(* IEC 61131-3 sources: POMIRTS_lab3/AS/Library/FB_lib, 3 files *)

(* ---- FB_lib.typ ---- *)
(********************************************************************
 * COPYRIGHT -- Bernecker + Rainer
 ********************************************************************
 * Library: FB_lib
 * File: FB_lib.typ
 * Author: B+R
 ********************************************************************
 * Data types of library FB_lib
 ********************************************************************)

TYPE
	FBDevice_typ : STRUCT			(*internal use*)
		MemorySize	: USINT ;
		DevAdress	: UDINT ;
		DevInfo	: UDINT ;
		Error	: UINT ;
		FBIdent	: UDINT ;
		DevNumber	: UINT ;
		DevType	: USINT ;
		ConfMsgNr	: USINT ;
		CommandMsgNr	: USINT ;
		StatusMsgNr	: USINT ;
		OtherMsgNr	: USINT ;
	END_STRUCT;
END_TYPE

(* ---- FB_lib.fun ---- *)
(********************************************************************
 * COPYRIGHT -- Bernecker + Rainer
 ********************************************************************
 * Library: FB_lib
 * File: FB_lib.fun
 * Author: B+R
 ********************************************************************
 * Functions and function blocks of library FB_lib
 ********************************************************************)

FUNCTION_BLOCK FBio					(*copies the input and output data areas between the B&R card and the specified buffers; asynchronous execution*)
	VAR_INPUT
		enable	:BOOL;				(*enables execution*)
		DevIdent	:UDINT;			(*device identifier returned from FBInit*)
		OutBuffer	:UDINT;			(*pointer to the output data area*)
		OutLen	:UDINT;				(*length of the output data area*)
		InBuffer	:UDINT;			(*pointer to the input data area*)
		InLen	:UDINT;				(*length of the input data area*)
	END_VAR
	VAR_OUTPUT
		status	:UINT;				(*execution status: ERR_OK, ERR_FUB_ENABLE_FALSE, ERR_FUB_BUSY, 0xXXXX = see help*)
	END_VAR
	VAR
		hmode	:USINT;				(*internal variable*)
	END_VAR
END_FUNCTION_BLOCK

FUNCTION_BLOCK FBStart				(*starts the I/O exchange process*)
	VAR_INPUT
		enable	:BOOL;				(*enables execution*)
		DevIdent	:UDINT;			(*device identifier returned from FBInit*)
	END_VAR
	VAR_OUTPUT
		status	:UINT;				(*execution status: ERR_OK, ERR_FUB_ENABLE_FALSE, 0xXXXX = see help*)
	END_VAR
END_FUNCTION_BLOCK

FUNCTION_BLOCK FBStop				(*stops the I/O exchange process*)
	VAR_INPUT
		enable	:BOOL;				(*enables execution*)
		DevIdent	:UDINT;			(*device identifier returned from FBInit*)
	END_VAR
	VAR_OUTPUT
		status	:UINT;				(*execution status: ERR_OK, ERR_FUB_ENABLE_FALSE, 0xXXXX = see help*)
	END_VAR
END_FUNCTION_BLOCK

FUNCTION_BLOCK FBSlaveStat			(*returns the current slave status*)
	VAR_INPUT
		enable	:BOOL;				(*enables execution*)
		DevIdent	:UDINT;			(*device identifier returned from FBInit*)
		SlaveReady	:UDINT;			(*pointer to a 16 byte array indicating whether a slave is in data transfer mode*)
		SlaveDiag	:UDINT;			(*pointer to a 16 byte array indicating the availability of diagnose information on slaves*)
	END_VAR
	VAR_OUTPUT
		status	:UINT;				(*execution status: ERR_OK, ERR_FUB_ENABLE_FALSE, 0xXXXX = see help*)
		SlaveStatus	:BOOL;			(*TRUE = a configured slave is not in data transfer mode or has diagnostic messages*)
	END_VAR
END_FUNCTION_BLOCK

FUNCTION_BLOCK FBInit				(*searches and initializes the specified device*)
	VAR_INPUT
		enable	:BOOL;				(*enables execution*)
		Device	:UDINT;				(*device name given as pointer, e.g., "SL2.SS1.IF1"*)
	END_VAR
	VAR_OUTPUT
		status	:UINT;				(*execution status: ERR_OK, ERR_FUB_ENABLE_FALSE, 0xXXXX = see help*)
		MemSize	:USINT;				(*indicates the FB size on the card*)
		DevIdent	:UDINT;			(*device identifier*)
		Run	:BOOL;					(*device in run: TRUE = in run, FALSE = not in run*)
		Configuration	:BOOL;		(*configuration: TRUE = valid, FALSE = not valid*)
	END_VAR
END_FUNCTION_BLOCK

FUNCTION_BLOCK FBSlaveExtStat		(*returns the exact status of a slave; asynchronous execution*)
	VAR_INPUT
		enable	:BOOL;				(*enables execution*)
		DevIdent	:UDINT;			(*device identifier returned from FBInit*)
		SlaveNumber	:USINT;			(*slave number*)
		SlaveDiagnostic	:UDINT;		(*pointer to an array of 48 bytes containing extended status and diagnostic information*)
	END_VAR
	VAR_OUTPUT
		status	:UINT;				(*execution status: ERR_OK, ERR_FUB_ENABLE_FALSE, ERR_FUB_BUSY, 0xXXXX = see help*)
		SlaveReady	:BOOL;			(*TRUE = slave is not in data transfer mode*)
		SlaveDiag	:BOOL;			(*TRUE = slave is in diagnostics mode*)
	END_VAR
	VAR
		istate	:UDINT;				(*internal variable*)
		waitCnt	:UINT;				(*internal variable*)
	END_VAR
END_FUNCTION_BLOCK

FUNCTION_BLOCK FBConfig				(*downloads the configuration; asynchronous execution*)
	VAR_INPUT
		enable	:BOOL;				(*enables execution*)
		DevIdent	:UDINT;			(*device identifier returned from FBInit*)
		ConfModulName	:UDINT;		(*configuration module name given as pointer*)
		Mode	:BOOL;				(*download mode, TRUE = sequential, FALSE = in one step*)
	END_VAR
	VAR_OUTPUT
		status	:UINT;				(*execution status: ERR_OK, ERR_FUB_ENABLE_FALSE, ERR_FUB_BUSY, 0xXXXX = see help*)
		Remaining	:UDINT;			(*displays the remaining segments until the configuration is completely loaded*)
	END_VAR
	VAR
		istate	:UDINT;				(*internal variable*)
		FileLength	:UINT;			(*internal variable*)
		waitCnt	:UINT;				(*internal variable*)
		OffsetCopy	:UDINT;			(*internal variable*)
		pData	:UDINT;				(*internal variable*)
		Ready	:USINT;				(*internal variable*)
		FirstMessage	:BOOL;		(*internal variable*)
		MsgPutReady	:BOOL;			(*internal variable*)
	END_VAR
END_FUNCTION_BLOCK

FUNCTION_BLOCK FBDialog				(*send messages to the B&R card; asynchronous execution*)
	VAR_INPUT
		enable	:BOOL;				(*enables execution*)
		DevIdent	:UDINT;			(*device identifier returned from FBInit*)
		Message	:UDINT;				(*pointer to the message structure*)
	END_VAR
	VAR_OUTPUT
		status	:UINT;				(*execution status: ERR_OK, ERR_FUB_ENABLE_FALSE, ERR_FUB_BUSY, 0xXXXX = see help*)
	END_VAR
	VAR
		istate	:UDINT;				(*internal variable*)
		tx	:USINT;					(*internal variable*)
		waitCount	:UINT;			(*internal variable*)
	END_VAR
END_FUNCTION_BLOCK

FUNCTION FBSearchDevices : UINT		(*searches the target system for B&R fieldbus cards*)
	VAR_INPUT
		pInfos	:UDINT;				(*pointer to the device information structure*)
		count	:USINT;				(*number of devices to be searched*)
	END_VAR
END_FUNCTION

FUNCTION_BLOCK FBGetMessage           (*sends a message to the B&R card and does not wait for an answer; asynchronous execution*)
	VAR_INPUT
		enable	:BOOL;                 (*enables execution*)
		DevIdent	:UDINT;            (*device identifier returned from DPMInit*)
		Message	:UDINT;                (*pointer to the message structure*)
	END_VAR
	VAR_OUTPUT
		status	:UINT;                 (*execution status: ERR_OK, ERR_FUB_ENABLE_FALSE, ERR_FUB_BUSY, 0xXXXX = see help*)
	END_VAR
	VAR
		waitCount	:UINT;             (*internal variable*)
	END_VAR
END_FUNCTION_BLOCK

FUNCTION_BLOCK FBPutMessage            (*reads out a message from the B&R card; asynchronous execution*)
	VAR_INPUT
		enable	:BOOL;                 (*enables execution*)
		DevIdent	:UDINT;            (*device identifier returned from DPMInit*)
		Message	:UDINT;                (*pointer to the message structure*)
	END_VAR
	VAR_OUTPUT
		status	:UINT;                 (*execution status: ERR_OK, ERR_FUB_ENABLE_FALSE, ERR_FUB_BUSY, 0xXXXX = see help*)
	END_VAR
	VAR
		waitCount	:UINT;             (*internal variable*)
	END_VAR
END_FUNCTION_BLOCK

(* ---- FB_lib.var ---- *)
(********************************************************************
 * COPYRIGHT -- Bernecker + Rainer
 ********************************************************************
 * Library: FB_lib
 * File: FB_lib.var
 * Author: B+R
 ********************************************************************
 * Local variables of library FB_lib
 ********************************************************************)

VAR CONSTANT
	FB_ERR_USR_MASTER_IS_STOPPED	: UINT	:= 12190;	(*master not in "RUN" state*)
	FB_ERR_USR_WRONG_HANDSHAKE	: UINT	:= 12191;		(*not supported handshake mode*)
	FB_ERR_USR_OUTLEN_TOO_LONG	: UINT	:= 12193;		(*cannot copy so much output data*)
	FB_ERR_USR_WRONG_DEVIDENT	: UINT	:= 12183;		(*invalid device identifier*)
	FB_ERR_USR_INLEN_TOO_LONG	: UINT	:= 12192;		(*cannot copy so much input data*)
	FB_ERR_USR_WRONG_MEMSIZE	: UINT	:= 12186;		(*specified memory size does not match device memory size*)
	FB_ERR_USR_DEV_MBOX_FULL	: UINT	:= 12180;		(*mailbox full*)
	FB_ERR_USR_WRONG_MODENR	: UINT	:= 12187;			(*specified mode number does not exist*)
	FB_ERR_USR_NOFREEIDENT	: UINT	:= 12185;			(*no more available identifier numbers for this device*)
	FB_host_reserved_flag	: USINT	:= 16;				(*internal constant*)
	FB_ERR_USR_SLAVE_CONF	: UINT	:= 12189;			(*specified slave not configured*)
	FB_ERR_USR_INTERNAL	: UINT	:= 12181;				(*internal error*)
	FB_ERR_USR_DATA_LNG	: UINT	:= 12188;				(*incorrect data length of configuration module*)
	FB_ERR_USR_BADIDENT	: UINT	:= 12184;				(*incorrect identifier number*)
	FB_ERR_USR_NOIDENT	: UINT	:= 12182;				(*no identifier number for the device*)
	FB_STATEACK_FLAG	: USINT	:= 8;					(*internal constant*)
	FB_NOTREADY_FLAG	: USINT	:= 32;					(*internal constant*)
	FB_HOSTACK_FLAG	: USINT	:= 1;						(*internal constant*)
	FB_DEVCOM_FLAG	: USINT	:= 2;						(*internal constant*)
	MAX_FB_BOARDS	: USINT	:= 8;						(*internal constant*)
	FB_RESET_FLAG	: USINT	:= 128;						(*internal constant*)
	FB_PDCOM_FLAG	: USINT	:= 4;						(*internal constant*)
	FB_INIT_FLAG	: USINT	:= 64;						(*internal constant*)
	FB_WORKING	: UINT	:= 65535;						(*function block still working*)
END_VAR
